FUNCTION_BLOCK AboutEqual
VAR_INPUT
	uiActual	: UINT;
	uiRequiered	: UINT;
	uiTolerance	: UINT;
END_VAR
VAR_OUTPUT
	OUT: BOOL;
END_VAR
VAR
	uiDifference: UINT;
END_VAR

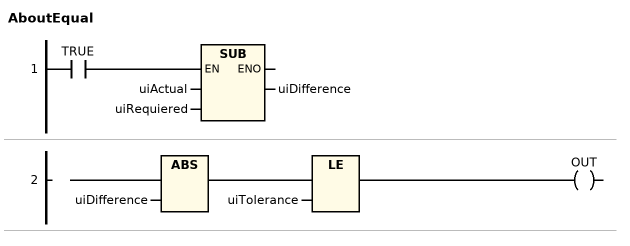
// NETWORK 1
uiDifference := uiActual - uiRequiered;

// NETWORK 2
OUT := ABS(uiDifference) <= uiTolerance;

END_FUNCTION_BLOCK

(* stored: Version 1.1.0.1, ProductVersion 3.1.4024.12
   POU AboutEqual: Id {87f40897-5c47-4545-a6b2-8b50610e3560}, SpecialFunc None *)
